{attribute 'pack_mode' := '1'}
TYPE ST_TcpTaskBuffer2 :
STRUCT
	BufferInfo : UDINT;
	TaskData : ST_TcpTask2;
END_STRUCT
END_TYPE

(* stored: Version 1.1.0.1, ProductVersion 3.1.4024.12
   DUT ST_TcpTaskBuffer2: Id {1840e779-4a10-4f35-9d96-bc6f6402e136} *)
